(* CoDeSys 2.3 export: Check48bool7SJ6xs0.EXP *)

(* POU SGL_Sismored/Sismored 4.0/Imported/Check48bool7SJ6xs0, ST *)
FUNCTION_BLOCK Check48bool7SJ6xs0
VAR_INPUT
	aValues : ARRAY [1..48] OF BOOL;
END_VAR
VAR_OUTPUT
	aMaskValues : ARRAY [1..48] OF BOOL;
	sTime: STRING;
END_VAR
VAR
	iN : INT;
	aLastValues : ARRAY[1..48] OF BOOL;
END_VAR
sTime := TimeAsString();

FOR iN := 1 TO 48 BY 1 DO
	IF aValues[iN] <> aLastValues[iN] THEN
		aMaskValues[iN] := TRUE;
	ELSE
		aMaskValues[iN] := FALSE;
	END_IF
END_FOR

aLastValues := aValues;
END_FUNCTION_BLOCK
